// TIA Portal V16 export
// export: Created 2024-12-03T15:41:45.4306822Z, ExportSetting WithReadOnly, DisplayName Totally Integrated Automation Portal, DisplayVersion V16 Update 6, DisplayName TIA Portal Version Control Interface, DisplayVersion V16 Update 2, DisplayName TIA Portal Openness, DisplayVersion V16 Update 6, DisplayName TIA Portal Teamcenter Gateway, DisplayVersion V16, DisplayName SINAMICS Startdrive Advanced, DisplayVersion V16 Update 5, DisplayName SINAMICS Startdrive G130, G150, S120, S150, SINAMICS MV, S210, DisplayVersion V16 Update 5, DisplayName SINAMICS Startdrive G110M, G120, G120C, G120D, G120P, G115D, DisplayVersion V16 Update 5, DisplayName STEP 7 Professional, DisplayVersion V16 Update 6, DisplayName STEP 7 Safety, DisplayVersion V16, DisplayName WinCC Advanced / Unified PC, DisplayVersion V16 Update 6
TYPE "G115D_OUTPUT_UDT"
// stored: CreationDate 2022-02-10T10:30:20.6863124Z, InterfaceModifiedDate 2021-08-10T11:24:29.0959269Z, IsConsistent true, LibraryConformanceStatus The object is library-conformant., ModifiedDate 2021-08-10T11:24:29.0959269Z
   STRUCT
      status : Struct
         CMD_DO24 : Bool;
         CMD_DO25 : Bool;
         ControlByPlc : Bool;
         SetPointInversed : Bool;
         spare_2 : Bool;
         MotPotSetPointRaise : Bool;
         MotPotSetPointLower : Bool;
         ParaMeterSet : Bool;
         on_off : Bool;
         NoCoastDown : Bool;
         NoQuickStop : Bool;
         EnableOperation : Bool;
         EnableRamp : Bool;
         EnableContinueRamp : Bool;
         EnableSetPoint : Bool;
         ackFault : Bool;
      END_STRUCT;
      setPointSpeed : Word;
   END_STRUCT;
END_TYPE
